Staubli VAL3: moveZ.pgx

public program moveZ(num nDz (dimensions=1))
  local frame frActual
  local point pFinal
  local point pHere
begin
  pHere=here(tActive,frActive)
  pFinal=compose(pHere,frActive,{0,0,nDz,0,0,0})
  movel(pFinal,tActive,mNomSpeed)
end
